{region '#Template'}
	{attribute 'Category' := 'Universal'}
	{attribute 'Version' := '0.0.1.0'}
	{attribute 'Tags' := 'Universal, Control, Scaling'}
	{attribute 'Description' := 'Skalierung	// Scaling'}
{endregion}
FUNCTION_BLOCK FB_BA_Scale_04 EXTENDS FB_BA_View
VAR_INPUT
	fX			: REAL;
END_VAR
VAR_OUTPUT
	fY			: REAL;
END_VAR
VAR_INPUT CONSTANT
	X1			: FB_BA_AV_Op;	
	X2			: FB_BA_AV_Op;	
	X3			: FB_BA_AV_Op;	
	X4			: FB_BA_AV_Op;	
	Y1			: FB_BA_AV_Op;	
	Y2			: FB_BA_AV_Op;
	Y3			: FB_BA_AV_Op;
	Y4			: FB_BA_AV_Op;
	YMin		: FB_BA_AV_Op;			
	YMax		: FB_BA_AV_Op;			
	Y			: FB_BA_AV_Op;		
END_VAR
VAR		
	Scale		: FB_BA_Chrct04;
END_VAR

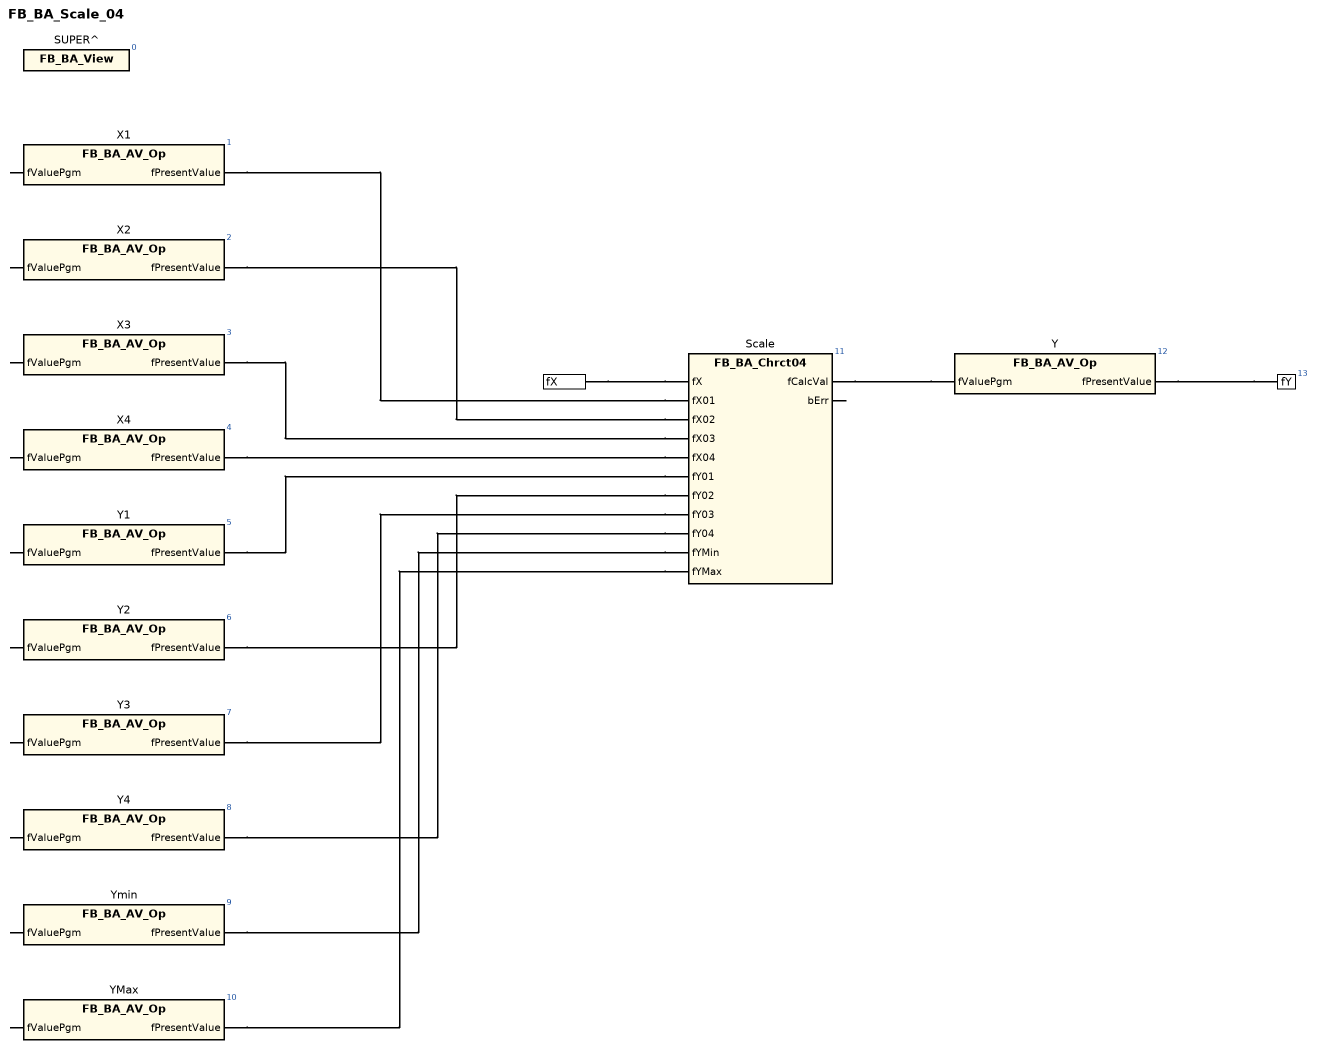
SUPER^(); // FB_BA_View
X1(); // FB_BA_AV_Op
X2(); // FB_BA_AV_Op
X3(); // FB_BA_AV_Op
X4(); // FB_BA_AV_Op
Y1(); // FB_BA_AV_Op
Y2(); // FB_BA_AV_Op
Y3(); // FB_BA_AV_Op
Y4(); // FB_BA_AV_Op
Ymin(); // FB_BA_AV_Op
YMax(); // FB_BA_AV_Op
Scale(
    fX := fX,
    fX01 := X1.fPresentValue,
    fX02 := X2.fPresentValue,
    fX03 := X3.fPresentValue,
    fX04 := X4.fPresentValue,
    fY01 := Y1.fPresentValue,
    fY02 := Y2.fPresentValue,
    fY03 := Y3.fPresentValue,
    fY04 := Y4.fPresentValue,
    fYMin := Ymin.fPresentValue,
    fYMax := YMax.fPresentValue); // FB_BA_Chrct04
Y(fValuePgm := Scale.fCalcVal); // FB_BA_AV_Op
fY := Y.fPresentValue;

METHOD FB_init : BOOL
VAR_INPUT
	bInitRetains : BOOL; // if TRUE, the retain variables are initialized (warm start / cold start)
	bInCopyCode : BOOL;  // if TRUE, the instance afterwards gets moved into the copy code (online change)
END_VAR
X1.iParent			:= THIS^;
X1.iLabel			:= LblUniControl.Scale_X01;	
X1.sObjectName		:= '{Idx=01}';								 	 
X1.eUnit			:= E_BA_Unit.eTemperature_DegreesCelsius;						 	 
X1.fValueRm			:= 15.0;
X1.fCOVIncrement	:= BA2_Param.fDefCOVIncrement;		

X2.iParent			:= THIS^;
X2.iLabel			:= LblUniControl.Scale_X02;							
X2.sObjectName		:= '{Idx=02}';								 	 
X2.eUnit			:= E_BA_Unit.eTemperature_DegreesCelsius;						 	 
X2.fValueRm			:= 0.0;
X2.fCOVIncrement	:= BA2_Param.fDefCOVIncrement;		

X3.iParent			:= THIS^;
X3.iLabel			:= LblUniControl.Scale_X03;	 						
X3.sObjectName		:= '{Idx=03}';								 	 
X3.eUnit			:= E_BA_Unit.eTemperature_DegreesCelsius;						 	 
X3.fValueRm			:= -10.0;
X3.fCOVIncrement	:= BA2_Param.fDefCOVIncrement;		

X4.iParent			:= THIS^;
X4.iLabel			:= LblUniControl.Scale_X04;						
X4.sObjectName		:= '{Idx=04}';								 	 
X4.eUnit			:= E_BA_Unit.eTemperature_DegreesCelsius;						 	 
X4.fValueRm			:= -20.0;
X4.fCOVIncrement	:= BA2_Param.fDefCOVIncrement;		

Y1.iParent			:= THIS^;
Y1.iLabel			:= LblUniControl.Scale_Y01;							
Y1.sObjectName		:= '{Idx=01}';								 	 
Y1.eUnit			:= E_BA_Unit.eTemperature_DegreesCelsius;						 	 
Y1.fValueRm			:= 25.0;
Y1.fCOVIncrement	:= BA2_Param.fDefCOVIncrement;		

Y2.iParent			:= THIS^;
Y2.iLabel			:= LblUniControl.Scale_Y02;				
Y2.sObjectName		:= '{Idx=02}';								 	 
Y2.eUnit			:= E_BA_Unit.eTemperature_DegreesCelsius;						 	 
Y2.fValueRm			:= 40.0;
Y2.fCOVIncrement	:= BA2_Param.fDefCOVIncrement;		

Y3.iParent			:= THIS^;
Y3.iLabel			:= LblUniControl.Scale_Y03;				
Y3.sObjectName		:= '{Idx=03}';								 	 
Y3.eUnit			:= E_BA_Unit.eTemperature_DegreesCelsius;						 	 
Y3.fValueRm			:= 55.0;
Y3.fCOVIncrement	:= BA2_Param.fDefCOVIncrement;		

Y4.iParent			:= THIS^;
Y4.iLabel			:= LblUniControl.Scale_Y04;				
Y4.sObjectName		:= '{Idx=04}';								 	 
Y4.eUnit			:= E_BA_Unit.eTemperature_DegreesCelsius;						 	 
Y4.fValueRm			:= 65.0;
Y4.fCOVIncrement	:= BA2_Param.fDefCOVIncrement;		

YMin.iParent		:= THIS^;
YMin.iLabel			:= LblUniControl.Scale_Ymin;		
YMin.sObjectName	:= '{Idx=01}';								 	 
YMin.eUnit			:= E_BA_Unit.eTemperature_DegreesCelsius;						 	 
YMin.fValueRm		:= 5.0;
YMin.fCOVIncrement	:= BA2_Param.fDefCOVIncrement;		

YMax.iParent		:= THIS^;
YMax.iLabel			:= LblUniControl.Scale_Ymax;			
YMax.sObjectName	:= '{Idx=01}';								 	 
YMax.eUnit			:= E_BA_Unit.eTemperature_DegreesCelsius;						 	 
YMax.fValueRm		:= 80.0;
YMax.fCOVIncrement	:= BA2_Param.fDefCOVIncrement;		

Y.iParent			:= THIS^;
Y.iLabel			:= LblUniControl.Scale_Y;				
Y.sObjectName		:= '{Idx=01}';								 	 
Y.eUnit				:= E_BA_Unit.eTemperature_DegreesCelsius;	
Y.fCOVIncrement		:= BA2_Param.fDefCOVIncrement;
END_METHOD

METHOD GetPoint : BOOL
VAR_INPUT
	nIndex		: INT;
END_VAR
VAR_OUTPUT
	fbObjectX	: I_BA_AnalogOpObject;
	fbObjectY	: I_BA_AnalogOpObject;
END_VAR
CASE (nIndex) OF
	1:
		fbObjectX := X1;
		fbObjectY := Y1;
	2:
		fbObjectX := X2;
		fbObjectY := Y2;
	3:
		fbObjectX := X3;
		fbObjectY := Y3;
	4:
		fbObjectX := X4;
		fbObjectY := Y4;
ELSE
	RETURN;
END_CASE

GetPoint := TRUE;
END_METHOD

END_FUNCTION_BLOCK

(* stored: Version 1.1.0.1, ProductVersion 3.1.4024.6
   POU FB_BA_Scale_04: Id {314bfc5a-1951-49d8-9f7d-d7251906fd70}, SpecialFunc None
   Folder Management: Id {8b2d3f0d-3623-48a1-afe6-9d9e4a036065}
   Method FB_init: Id {c6dd6d21-4b56-4c83-8ff8-7962632c988b}
   Method GetPoint: Id {0fab3497-63cf-4be3-8934-74fb55739000} *)
